// TwinCAT 3 PLC project Simple_Factory_Pattern
// ProgramVersion: 3.1.4024.0
// libraries:
//   Tc2_Standard, * (Beckhoff Automation GmbH)
//   Tc2_System, * (Beckhoff Automation GmbH)
//   Tc3_DynamicMemory, * (Beckhoff Automation GmbH)
//   Tc3_Module, * (Beckhoff Automation GmbH)
//   Tc3_UnitTest, * (Zerlauth)
// project tree:
//   Class/ EtherCATDevice.TcPOU (not stored), I_EtherCATDevice.TcIO
//   Simple Factory/ EtherCATFactory.TcPOU
//   / PlcTask.TcTTO (not stored)
//   POUs/ MAIN.TcPOU
// real-time tasks:
//   TASK PlcTask: cycle T#10ms, priority 20, ADS port 350
//   TASK PlcTask1: cycle T#10ms, priority 21, ADS port 351
//   TASK PlcTask2: cycle T#10ms, priority 22, ADS port 352
//   TASK PlcTask3: cycle T#10ms, priority 23, ADS port 353
//   TASK PlcTask4: cycle T#10ms, priority 24, ADS port 354
//   TASK PlcTask5: cycle T#10ms, priority 25, ADS port 355
//   TASK PlcTask6: cycle T#10ms, priority 26, ADS port 356
//   TASK PlcTask7: cycle T#10ms, priority 27, ADS port 357
//   TASK PlcTask8: cycle T#10ms, priority 28, ADS port 358
//   TASK PlcTask9: cycle T#10ms, priority 29, ADS port 359
//   TASK PlcTask10: cycle T#10ms, priority 30, ADS port 360
//   TASK PlcTask11: cycle T#10ms, priority 31, ADS port 361

// ---- Class/I_EtherCATDevice.TcIO
INTERFACE I_EtherCATDevice

METHOD IsDeviceOK : BOOL
VAR_INPUT
END_VAR
END_METHOD

END_INTERFACE

// ---- Simple Factory/EtherCATFactory.TcPOU
FUNCTION_BLOCK EtherCATFactory
VAR

END_VAR

METHOD PUBLIC CreateEtherCATDevice : I_EtherCATDevice
VAR_INPUT
END_VAR

VAR
	devicePtr: POINTER TO EtherCATDevice;
END_VAR
devicePtr := __NEW(EtherCATDevice);
CreateEtherCATDevice := devicePtr^;
END_METHOD

END_FUNCTION_BLOCK

// ---- POUs/MAIN.TcPOU
PROGRAM MAIN
VAR
	EtherCATIOFactory : EtherCATFactory;
	GetEtherCATDevice: BOOL;
	myDevcie : I_EtherCATDevice;
	CheckMyDevice: BOOL;
	value: BOOL;
END_VAR

IF GetEtherCATDevice THEN
	GetEtherCATDevice := FALSE;
	myDevcie := EtherCATIOFactory.CreateEtherCATDevice();
END_IF

IF CheckMyDevice THEN
	CheckMyDevice := false;
    value := myDevcie.IsDeviceOK();
END_IF

END_PROGRAM
